FUNCTION_BLOCK EmergencyRecipeSequenceSludgeBuffer (* Basic Function Block Type *)
  (* Standard: 61499-2 *)
  (* Version 0.0, 7/4/2026, Schneider Electric, Template *)
  PACKAGE SE.Nereda;
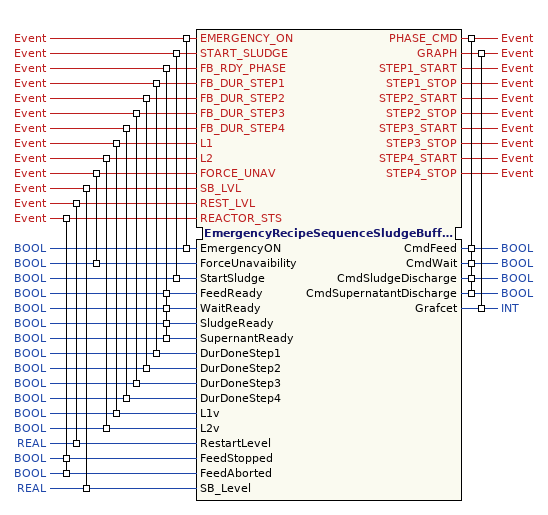
  EVENT_INPUT
    EMERGENCY_ON WITH EmergencyON;
    START_SLUDGE WITH StartSludge;
    FB_RDY_PHASE WITH FeedReady, SupernantReady, SludgeReady, WaitReady;
    FB_DUR_STEP1 WITH DurDoneStep1;
    FB_DUR_STEP2 WITH DurDoneStep2;
    FB_DUR_STEP3 WITH DurDoneStep3;
    FB_DUR_STEP4 WITH DurDoneStep4;
    L1 WITH L1v;
    L2 WITH L2v;
    FORCE_UNAV WITH ForceUnavaibility;
    SB_LVL WITH SB_Level;
    REST_LVL WITH RestartLevel;
    REACTOR_STS WITH FeedStopped, FeedAborted;
  END_EVENT
  EVENT_OUTPUT
    PHASE_CMD WITH CmdFeed, CmdSupernatantDischarge, CmdSludgeDischarge, CmdWait;
    GRAPH WITH Grafcet;
    STEP1_START;
    STEP1_STOP;
    STEP2_START;
    STEP2_STOP;
    STEP3_START;
    STEP3_STOP;
    STEP4_START;
    STEP4_STOP;
  END_EVENT
  VAR_INPUT
    EmergencyON : BOOL;
    ForceUnavaibility : BOOL;
    StartSludge : BOOL;
    FeedReady : BOOL;
    WaitReady : BOOL;
    SludgeReady : BOOL;
    SupernantReady : BOOL;
    DurDoneStep1 : BOOL;
    DurDoneStep2 : BOOL;
    DurDoneStep3 : BOOL;
    DurDoneStep4 : BOOL;
    L1v : BOOL;
    L2v : BOOL;
    RestartLevel : REAL;
    FeedStopped : BOOL;
    FeedAborted : BOOL;
    SB_Level : REAL;
  END_VAR
  VAR_OUTPUT
    CmdFeed : BOOL;
    CmdWait : BOOL;
    CmdSludgeDischarge : BOOL;
    CmdSupernatantDischarge : BOOL;
    Grafcet : INT;
  END_VAR
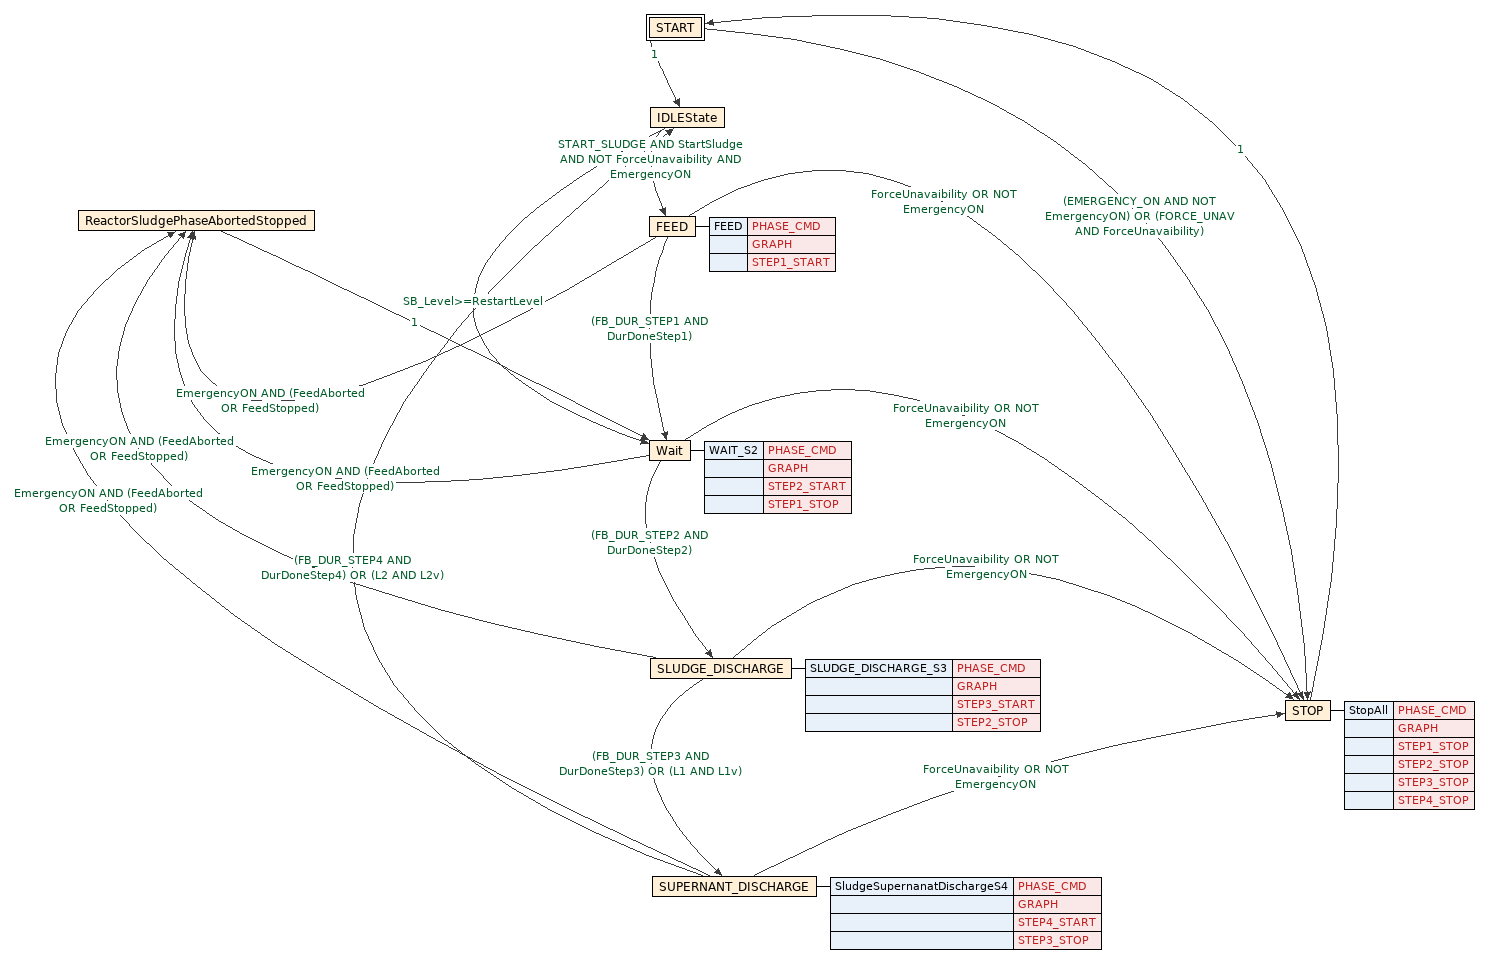
  EC_STATES
    START; (* Initial State *)
    FEED : FEED -> PHASE_CMD, -> GRAPH, -> STEP1_START;
    Wait : WAIT_S2 -> PHASE_CMD, -> GRAPH, -> STEP2_START, -> STEP1_STOP;
    SLUDGE_DISCHARGE : SLUDGE_DISCHARGE_S3 -> PHASE_CMD, -> GRAPH, -> STEP3_START, -> STEP2_STOP;
    SUPERNANT_DISCHARGE : SludgeSupernanatDischargeS4 -> PHASE_CMD, -> GRAPH, -> STEP4_START, -> STEP3_STOP;
    STOP : StopAll -> PHASE_CMD, -> GRAPH, -> STEP1_STOP, -> STEP2_STOP, -> STEP3_STOP, -> STEP4_STOP;
    IDLEState;
    ReactorSludgePhaseAbortedStopped;
  END_STATES
  EC_TRANSITIONS
    IDLEState TO FEED := START_SLUDGE AND StartSludge AND NOT ForceUnavaibility AND EmergencyON;
    FEED TO Wait := (FB_DUR_STEP1 AND DurDoneStep1);
    Wait TO SLUDGE_DISCHARGE := (FB_DUR_STEP2 AND DurDoneStep2);
    SLUDGE_DISCHARGE TO SUPERNANT_DISCHARGE := (FB_DUR_STEP3 AND DurDoneStep3) OR (L1 AND L1v);
    SUPERNANT_DISCHARGE TO IDLEState := (FB_DUR_STEP4 AND DurDoneStep4) OR (L2 AND L2v);
    START TO STOP := (EMERGENCY_ON AND NOT EmergencyON) OR (FORCE_UNAV AND ForceUnavaibility);
    STOP TO START := 1;
    FEED TO STOP := ForceUnavaibility OR NOT EmergencyON;
    Wait TO STOP := ForceUnavaibility OR NOT EmergencyON;
    SLUDGE_DISCHARGE TO STOP := ForceUnavaibility OR NOT EmergencyON;
    SUPERNANT_DISCHARGE TO STOP := ForceUnavaibility OR NOT EmergencyON;
    IDLEState TO Wait := SB_Level>=RestartLevel;
    START TO IDLEState := 1;
    ReactorSludgePhaseAbortedStopped TO Wait := 1;
    SUPERNANT_DISCHARGE TO ReactorSludgePhaseAbortedStopped := EmergencyON AND (FeedAborted OR FeedStopped);
    SLUDGE_DISCHARGE TO ReactorSludgePhaseAbortedStopped := EmergencyON AND (FeedAborted OR FeedStopped);
    FEED TO ReactorSludgePhaseAbortedStopped := EmergencyON AND (FeedAborted OR FeedStopped);
    Wait TO ReactorSludgePhaseAbortedStopped := EmergencyON AND (FeedAborted OR FeedStopped);
  END_TRANSITIONS
  ALGORITHM FEED IN ST:
;
CmdFeed := TRUE;
CmdWait := FALSE;
CmdSludgeDischarge := FALSE;
CmdSupernatantDischarge := FALSE;

Grafcet := 1;
  END_ALGORITHM
  ALGORITHM StopAll IN ST:
;
CmdFeed := FALSE;
CmdWait := FALSE;
CmdSludgeDischarge := FALSE;
CmdSupernatantDischarge := FALSE;

Grafcet := 5;
  END_ALGORITHM
  ALGORITHM WAIT_S2 IN ST:
;
CmdFeed := FALSE;
CmdWait := TRUE;
CmdSludgeDischarge := FALSE;
CmdSupernatantDischarge := FALSE;

Grafcet := 2;
  END_ALGORITHM
  ALGORITHM SLUDGE_DISCHARGE_S3 IN ST:
;
CmdFeed := FALSE;
CmdWait := FALSE;
CmdSludgeDischarge := TRUE;
CmdSupernatantDischarge := FALSE;

Grafcet := 3;
  END_ALGORITHM
  ALGORITHM SludgeSupernanatDischargeS4 IN ST:
;
CmdFeed := FALSE;
CmdWait := FALSE;
CmdSludgeDischarge := FALSE;
CmdSupernatantDischarge := TRUE;

Grafcet := 4;
  END_ALGORITHM
END_FUNCTION_BLOCK
